{attribute 'linkalways'} 
{attribute 'no_explicit_call' := 'This FB is a CLASS and must be accessed using methods or properties'}
{attribute 'enable_dynamic_creation'}
FUNCTION_BLOCK _ETcVnFindTemplateWalshOptions EXTENDS EnumDatatypeBase
VAR
	localData : ETcVnFindTemplateWalshOptions;
	activeData : REFERENCE TO ETcVnFindTemplateWalshOptions;
	enumBaseDatatype : _UDINT(localData);
END_VAR

METHOD PRIVATE AddLocalEnumeration
VAR_INPUT
	Enumeration : T_MAXSTRING;
	Value : ETcVnFindTemplateWalshOptions;
END_VAR
AddEnumeration(Enumeration, Value);
END_METHOD

PROPERTY PUBLIC Address : PVOID
GET
Address := ADR(activeData);
END_GET
END_PROPERTY

METHOD PUBLIC ClearReference
VAR_INPUT
END_VAR
activeData REF= localData;
SetBaseDatatypeReference();
END_METHOD

METHOD PUBLIC Clone : I_Datatype
VAR
    pClone : POINTER TO _ETcVnFindTemplateWalshOptions;
END_VAR
pClone := __NEW(_ETcVnFindTemplateWalshOptions(InitialValue := Value));
Clone := pClone^;
END_METHOD

METHOD FB_init : BOOL
VAR_INPUT
	bInitRetains : BOOL; // if TRUE, the retain variables are initialized (warm start / cold start)
	bInCopyCode : BOOL;  // if TRUE, the instance afterwards gets moved into the copy code (online change)
	InitialValue : ETcVnFindTemplateWalshOptions;
END_VAR
localData := InitialValue;
AddBaseDatatype(enumBaseDatatype);
ClearReference();

AddLocalEnumeration('TCVN_FTWO_NONE', ETcVnFindTemplateWalshOptions.TCVN_FTWO_NONE);
AddLocalEnumeration('TCVN_FTWO_SKIP_DC', ETcVnFindTemplateWalshOptions.TCVN_FTWO_SKIP_DC);
AddLocalEnumeration('TCVN_FTWO_WD_STOP_CORRECTION', ETcVnFindTemplateWalshOptions.TCVN_FTWO_WD_STOP_CORRECTION);
AddLocalEnumeration('TCVN_FTWO_FUSE_MATCHES', ETcVnFindTemplateWalshOptions.TCVN_FTWO_FUSE_MATCHES);
AddLocalEnumeration('TCVN_FTWO_ROTATED_RECTANGLE', ETcVnFindTemplateWalshOptions.TCVN_FTWO_ROTATED_RECTANGLE);
AddLocalEnumeration('TCVN_FTWO_MATCH_OPPOSITE_RANGE', ETcVnFindTemplateWalshOptions.TCVN_FTWO_MATCH_OPPOSITE_RANGE);
END_METHOD

PROPERTY PUBLIC Identifier : T_MAXSTRING
GET
Identifier := 'ETcVnFindTemplateWalshOptions';
END_GET
END_PROPERTY

METHOD IsEnumeratorValueEqual : BOOL
VAR_INPUT
	Enumerator : I_KeyValueForwardEnumerator;
END_VAR
VAR
	storedValue : ETcVnFindTemplateWalshOptions;
END_VAR
IF NOT Enumerator.TryGet(storedValue) THEN
	RETURN;
END_IF

IsEnumeratorValueEqual := storedValue = activeData;
END_METHOD

METHOD PUBLIC MakeReferenceTo
VAR_INPUT
	ReferenceTarget : REFERENCE TO ETcVnFindTemplateWalshOptions;
END_VAR
activeData REF= ReferenceTarget;
SetBaseDatatypeReference();
END_METHOD

METHOD PROTECTED SetBaseDatatypeReference
VAR_INPUT
END_VAR
enumBaseDatatype.MakeReferenceTo(activeData);
END_METHOD

PROPERTY PUBLIC Size : UDINT
GET
Size := SIZEOF(activeData);
END_GET
END_PROPERTY

METHOD TryMakeReferenceTo : BOOL
VAR_INPUT
	Target : I_Datatype;
END_VAR
VAR
	pTargetData : POINTER TO ETcVnFindTemplateWalshOptions;
END_VAR
IF NOT IsEquivalentTo(Target) THEN
	RETURN;
END_IF

pTargetData := Target.Address;
activeData REF= pTargetData^;
SetBaseDatatypeReference();
TryMakeReferenceTo := TRUE;
END_METHOD

PROPERTY PUBLIC Value : ETcVnFindTemplateWalshOptions
GET
Value := activeData;
END_GET
SET
activeData := Value;
END_SET
END_PROPERTY

END_FUNCTION_BLOCK

(* stored: Version 1.1.0.1, ProductVersion 3.1.4026.13
   POU _ETcVnFindTemplateWalshOptions: Id {3c39b9af-46bb-03c6-2fd5-10fd28d55341}, SpecialFunc None
   Folder Core: Id {fcf3e7ce-5114-05ce-3984-17002024e200}
   Folder Protected: Id {c04e1a13-0bfb-0eae-0e38-3b7a50cf2961}
   Folder Customize: Id {a5a8c0d2-7e3b-0410-309b-c58ee0ee52f2}
   Folder Constructor: Id {5cf6fc11-f298-0107-134e-1bedd731048f}
   Folder Private: Id {76edd914-5aa1-092b-3178-3d54106f461f}
   Folder Protected: Id {1b55dd5a-1f2c-08d2-2513-d2f8f2abe84c}
   Method AddLocalEnumeration: Id {438a5697-3d6b-0639-124c-494a6ffd9e70}
   Property Address: Id {d36759ca-2555-0e67-36d5-9adfe9f2367a}
   Get Get: Id {f90672fe-a030-0e70-05ee-fbf861f76321}
   Method ClearReference: Id {d1cb0eae-ed62-0535-38bb-d543665facad}
   Method Clone: Id {8bf5adf8-fcbe-083f-0cc5-4d041fd621bc}
   Method FB_init: Id {1717f5a9-268c-0a67-2252-8a86b40b5a89}
   Property Identifier: Id {2cdc1024-fda7-0056-16d1-b89a762791e9}
   Get Get: Id {17be8dab-5c7e-0fdb-1ae9-ad6d6ae4f6b7}
   Method IsEnumeratorValueEqual: Id {aaf4b3d4-cc43-016e-2e13-d286b485506c}
   Method MakeReferenceTo: Id {790fa42c-8dcf-025e-0255-3bceb1931d67}
   Method SetBaseDatatypeReference: Id {f703d347-16b1-092a-2a2c-68d3abb0a7ca}
   Property Size: Id {6d25dcb1-af39-0bef-2a27-0b49d8c47ba7}
   Get Get: Id {14ef0eb6-8fa3-0e2a-02a9-6756e848ecac}
   Method TryMakeReferenceTo: Id {d18ea075-9a88-0c2a-02f0-f2db3bc75989}
   Property Value: Id {8e8cec71-bd93-01f9-025c-a99f6fd17ea2}
   Get Get: Id {45ec0a08-2b67-0cb8-2e69-35e0b4ab98f0}
   Set Set: Id {74954d65-72b5-065d-3cd0-68ae0c4bf3b9} *)
